FUNCTION_BLOCK RunCylinder Extends ExecuteBase
VAR			

	COMMAND_CACHED : eCylinderCommands; //1 , HMI->PLC
	LAST_COMMAND : eCylinderCommands;   //2 , 
		
	ACT_A AT %Q* : ARRAY[1..2] OF BOOL;
	ACT_B AT %Q* : ARRAY[1..2] OF BOOL;
	
	SENSOR_A AT %I* : ARRAY[1..4] OF BOOL;
	SENSOR_B AT %I* : ARRAY[1..4] OF BOOL;

	nCounter : INT := 0;
	bMatched : BOOL := false;
		
	BIT_WARNING : BIT; //0
	BIT_A_MATCH : BIT; //1
	BIT_B_MATCH : BIT; //2
	BIT_WARN_SUPPRESS : BIT; //3 , (Control)
	
	BIT_DONE : BIT; //5
	
END_VAR
VAR PERSISTENT
	A_SENSOR_USED_COUNT : INT := 0;
	B_SENSOR_USED_COUNT : INT :=0 ;		

	TMR_WATCH_DOG : TON ; //Watch dog timer
	TMR_DELAY_TO_A : TON;
	TMR_DELAY_TO_B : TON;
END_VAR

SUPER^();

//Run timers
TMR_WATCH_DOG(IN:= , PT:= , Q=> , ET=> );
TMR_DELAY_TO_A(IN:= , PT:= , Q=> , ET=> );
TMR_DELAY_TO_B(IN:= , PT:= , Q=> , ET=> );

// scan all sensor status
BIT_A_MATCH := TRUE;
FOR nCounter := 1 TO A_SENSOR_USED_COUNT BY 1 DO
	BIT_A_MATCH := (BIT_A_MATCH AND SENSOR_A[nCounter]);
END_FOR
BIT_B_MATCH := TRUE;
FOR nCounter := 1 TO B_SENSOR_USED_COUNT BY 1 DO
	BIT_B_MATCH := (BIT_B_MATCH AND SENSOR_B[nCounter]);
END_FOR

// if watch dog had been reset due to command changed in previous scan
// restart
//IF NOT TMR_WATCH_DOG.IN THEN
//	TMR_WATCH_DOG.IN := TRUE;
//END_IF

// once command changes , reset timer counter
IF COMMAND_CACHED <> LAST_COMMAND THEN
	TMR_DELAY_TO_A.IN := (COMMAND_CACHED=eCylinderCommands.COMMAND_A); //active A delay timer
	TMR_DELAY_TO_B.IN := (COMMAND_CACHED=eCylinderCommands.COMMAND_B); //if no sensor B , active B delay timer
	
	//reset done/warn
	BIT_DONE := FALSE;
	BIT_WARNING := FALSE;
	
	//output process , for nuetual command , hold current position
	IF COMMAND_CACHED <> eCylinderCommands.NO_COMMAND THEN
		FOR nCounter:=1 TO 2 BY 1 DO
			ACT_A[nCounter] := (COMMAND_CACHED = eCylinderCommands.COMMAND_A);
			ACT_B[nCounter] := (COMMAND_CACHED = eCylinderCommands.COMMAND_B);
		END_FOR
	END_IF
	
END_IF


//reset
bMatched := FALSE;
// Check if match
CASE COMMAND_CACHED OF
	eCylinderCommands.NO_COMMAND:
	bMatched:= TRUE;
	
	eCylinderCommands.COMMAND_A:
	IF TMR_DELAY_TO_A.Q THEN
		bMatched:= (BIT_A_MATCH OR (A_SENSOR_USED_COUNT=0)) AND ((NOT BIT_B_MATCH) OR (B_SENSOR_USED_COUNT=0));
	END_IF
	
	eCylinderCommands.COMMAND_B:
	IF TMR_DELAY_TO_B.Q THEN
		bMatched:= ((NOT BIT_A_MATCH) OR (A_SENSOR_USED_COUNT=0)) AND (BIT_B_MATCH OR (B_SENSOR_USED_COUNT=0) );
	END_IF
		
END_CASE

//start
IF NOT bMatched AND (TMR_DELAY_TO_B.Q OR TMR_DELAY_TO_A.Q) THEN
	TMR_WATCH_DOG.in := TRUE;
ELSE
	TMR_WATCH_DOG.in := FALSE;
END_IF

// status update
BIT_DONE := bMatched OR (NOT bMatched AND (BIT_WARN_SUPPRESS OR isShutVerification) AND TMR_WATCH_DOG.Q);
BIT_WARNING := (NOT bMatched) AND (NOT BIT_WARN_SUPPRESS) AND TMR_WATCH_DOG.Q AND (TMR_DELAY_TO_B.Q OR TMR_DELAY_TO_A.Q);


// cache last command
LAST_COMMAND := COMMAND_CACHED;

//scan-out status
//comm.STATUS_WORD.0 := BIT_WARNING;
//comm.STATUS_WORD.1 := BIT_A_MATCH;
//comm.STATUS_WORD.2 := BIT_B_MATCH;
//comm.STATUS_WORD.5 := BIT_DONE;

METHOD ConfigureRead : CellDataBlock
VAR_INPUT
	input : CellDataBlock; //would offer sub-index ...etc
	mode : eModes;
END_VAR

ConfigureRead.cylinder.sensorAUsedCount := TO_WORD(A_SENSOR_USED_COUNT);
ConfigureRead.cylinder.sensorBUsedCount := TO_WORD(B_SENSOR_USED_COUNT);

ConfigureRead.cylinder.timerSetValue := TO_WORD(TMR_WATCH_DOG.PT);
ConfigureRead.cylinder.timerSetValue := TO_WORD(TMR_DELAY_TO_A.PT);
ConfigureRead.cylinder.timerSetValue := TO_WORD(TMR_DELAY_TO_B.PT);
END_METHOD

METHOD ConfigureWrite : BOOL
VAR_INPUT
	input : CellDataBlock;
	mode : eModes;
END_VAR
A_SENSOR_USED_COUNT := TO_INT(input.cylinder.sensorAUsedCount);
B_SENSOR_USED_COUNT := TO_INT(input.cylinder.sensorBUsedCount);

TMR_WATCH_DOG.PT := TO_TIME(input.cylinder.timerSetValue);
TMR_DELAY_TO_A.PT := TO_TIME(input.cylinder.timerSetValue);
TMR_DELAY_TO_B.PT := TO_TIME(input.cylinder.timerSetValue);
END_METHOD

METHOD Control : BOOL
VAR_INPUT
	input : CellDataBlock;
	mode : eModes;
END_VAR
Execute(argCommand:= input.cylinder.command);
Control:=true;
END_METHOD

METHOD ErrorClear : BOOL
VAR_INPUT
	input : eErrorClearWays;
END_VAR
CASE input OF
	eErrorClearWays.RESET:
		//Timer reset only
	eErrorClearWays.IGNORE:
		//suppress warning
		BIT_WARN_SUPPRESS := TRUE;
END_CASE
END_METHOD

METHOD ErrorDetect : UDINT
VAR_INPUT
END_VAR
ErrorDetect := 0;
IF BIT_WARNING THEN
	ErrorDetect := COMMAND_CACHED; //distinguish different error 
END_IF
END_METHOD

METHOD Execute : BOOL
VAR_INPUT
	argCommand : eCylinderCommands;
END_VAR
VAR
	outDone  : BOOL ;
END_VAR
// store command
COMMAND_CACHED := argCommand;

outDone := BIT_DONE AND NOT BIT_WARNING AND (COMMAND_CACHED = LAST_COMMAND);

//reset surpress
IF outDone THEN
	BIT_WARN_SUPPRESS := FALSE;
END_IF

Execute:=outDone; //return
END_METHOD

METHOD FB_init : BOOL
VAR_INPUT
	bInitRetains : BOOL; // if TRUE, the retain variables are initialized (warm start / cold start)
	bInCopyCode : BOOL;  // if TRUE, the instance afterwards gets moved into the copy code (online change)
	
	//argASensorUsed : INT := 0;
	//argBSensorUsed : INT := 0;
END_VAR
//A_SENSOR_USED_COUNT := argASensorUsed;
//B_SENSOR_USED_COUNT := argBSensorUsed;

//given timer initial value
//TMR_WATCH_DOG.PT := T#200MS;
//TMR_DELAY_TO_A.PT := T#200MS;
//TMR_DELAY_TO_B.PT := T#200MS;
IF bInitRetains THEN
	TMR_WATCH_DOG.PT := T#200MS;
	TMR_DELAY_TO_A.PT := T#200MS;
	TMR_DELAY_TO_B.PT := T#200MS;
END_IF
END_METHOD

METHOD Monitor : CellDataBlock
VAR_INPUT
END_VAR
VAR CONSTANT
	bit0Warn : INT :=0;
	bit1MonGroupA : INT :=1;
	bit2MonGroupB : INT :=2;
	bit3CtlSuppress : INT :=3;
	bit4TmrOn : INT :=4;
	bit5Done : INT := 5;
	//New
	bit6TmrAOn : INT :=6;
	bit7TmrBOn : INT :=7;
END_VAR
Monitor.cylinder.statusWord.bit0Warn := BIT_WARNING;
Monitor.cylinder.statusWord.bit1MonGroupA := BIT_A_MATCH;
Monitor.cylinder.statusWord.bit2MonGroupB := BIT_B_MATCH;
Monitor.cylinder.statusWord.bit3CtlSuppress := BIT_WARN_SUPPRESS;
Monitor.cylinder.statusWord.bit4TmrOn := TMR_WATCH_DOG.Q;
Monitor.cylinder.statusWord.bit5Done := BIT_DONE;

Monitor.cylinder.statusWord.bit6TmrAOn := TMR_DELAY_TO_A.Q;
Monitor.cylinder.statusWord.bit7TmrBOn := TMR_DELAY_TO_B.Q;

Monitor.cylinder.lastCommand := LAST_COMMAND;
END_METHOD

METHOD TypeCode : eCategrories
VAR_INPUT
END_VAR
TypeCode := eCategrories.SELECTION_CYLINDER;
END_METHOD

END_FUNCTION_BLOCK

(* stored: Version 1.1.0.1, ProductVersion 3.1.4024.0
   POU RunCylinder: Id {a99bf5d1-aaa3-4095-9742-005d9ab3fed8}, SpecialFunc None
   Folder CommonBase: Id {48bea1d3-0a28-439a-92dd-8f8417445059}
   Method ConfigureRead: Id {bc98ac9f-d51a-43ad-b528-a1a54fe67ea0}
   Method ConfigureWrite: Id {f3b24b0b-d22d-4018-b1c9-709a957955d9}
   Method Control: Id {57e57159-f3d2-45e6-85f3-9a286c6e359d}
   Method ErrorClear: Id {945c9ccd-86db-44c6-8d20-e9e7b141f3bf}
   Method ErrorDetect: Id {6a0ed216-b71b-4070-ba95-2d84d65ddbd3}
   Method Execute: Id {13693201-8c27-444e-bbfc-9d5e6a727077}
   Method FB_init: Id {41827ab5-0173-413a-8bd3-19090e017f80}
   Method Monitor: Id {120aac0f-3608-4cae-b6d2-bb459b1d4cf7}
   Method TypeCode: Id {2fbd4fdf-fcb0-4d45-95f6-2e5788341375} *)
